FUNCTION "LHTTP_ExtractStringFromArray" : Word   // FC2, SCL
{ S7_Optimized_Access := 'TRUE' }
VERSION : 0.1
   VAR_INPUT
      textBefore : String;   // Text before text that is extracted
      textAfter : String;   // Text after text that is extracted
   END_VAR
   VAR_OUTPUT
      extractedString : String;   // Extracted string
   END_VAR
   VAR_IN_OUT
      searchIn : Array[*] of Char;   // Array of Char to search in
   END_VAR
   VAR_TEMP
      tempLowerBound : DInt;   // Lower bound of given array
      tempNumElements : UDInt;   // Number of elements in given array
      tempPosInArray : DInt;   // Position in array during search
      tempLenTextBefore : Int;   // Length of text before
      tempPosTextBefore : DInt;   // Position of text before in array of Char
      tempLenTextAfter : Int;   // Length of text after
      tempPosTextAfter : Int;   // Position of text after in converted string
      tempString : String;   // Temporary string to work with
   END_VAR
   // Ret_Val : Return value; 16#0000: Successful, text was found, 16#9001: Unsuccessful, only start text was found, extracted String is filled with characters after start text, 16#9002: Unsuccessful, neither text was found
   VAR CONSTANT
      LEN_STRING : UInt := 254;   // Max. length of String
      STATUS_TEXT_FOUND : Word := 16#0000;   // Texts before and after were found
      STATUS_ONLY_START : Word := 16#9001;   // Only text before was found
      STATUS_NOTHING_FOUND : Word := 16#9002;   // Neither text was found
   END_VAR
BEGIN
   //=============================================================================
   // SIEMENS AG
   // (c)Copyright 2019
   //-----------------------------------------------------------------------------
   // Library:       LHTTP
   // Tested with:   CPU 1516-3 PN/DP V2.6
   // Engineering:   TIA Portal V15.1
   // Restrictions:  --
   // Requirements:  --
   // Functionality: Extracts a String specified by a text before and after
   //                from an array of Char
   //-----------------------------------------------------------------------------
   // Change log table:
   // Version    Date         Expert in charge         Changes applied
   // 01.00.00   01.04.2019   Siemens Online Support   First released version
   //=============================================================================

   // Initialization
   #tempPosTextBefore := 0;
   #tempPosTextAfter := 0;
   #tempLenTextBefore := LEN(#textBefore);
   #tempLenTextAfter := LEN(#textAfter);
   #extractedString := '';
   #LHTTP_ExtractStringFromArray := #STATUS_NOTHING_FOUND;

   // Get number of elements
   #tempPosInArray := #tempLowerBound := LOWER_BOUND(ARR := #searchIn, DIM := 1);
   #tempNumElements := DINT_TO_UDINT(UPPER_BOUND(ARR := #searchIn, DIM := 1) - #tempLowerBound + 1);


   // Search for text before until something was found
   REPEAT

     // Convert Chars to String
     Chars_TO_Strg(Chars  := #searchIn,
                   pChars := #tempPosInArray - #tempLowerBound, // Subtract offset since pChars is zero based
                   Cnt    := UDINT_TO_UINT(MIN(IN1 := #LEN_STRING, IN2 := #tempNumElements)),
                   Strg   => #tempString);

     // Search for text before
     #tempPosTextBefore := FIND(IN1 := #tempString, IN2 := #textBefore);

     // Text before was found
     IF #tempPosTextBefore > 0 THEN

       // Set position in array to end of text before
       #tempPosInArray += #tempPosTextBefore + #tempLenTextBefore - 1;

       // Create new string from end of text before
       Chars_TO_Strg(Chars  := #searchIn,
                     pChars := #tempPosInArray - #tempLowerBound, // Subtract offset since pChars is zero based
                     Cnt    := UDINT_TO_UINT(MIN(IN1 := #LEN_STRING, IN2 := #tempNumElements)),
                     Strg   => #tempString);

       // Find end of string to be extracted
       #tempPosTextAfter := FIND(IN1 := #tempString, IN2 := #textAfter);

       IF #tempPosTextAfter > 0 THEN // Shorten string if text after was found

         #extractedString := LEFT(IN := #tempString, L := #tempPosTextAfter - 1);
         #LHTTP_ExtractStringFromArray := #STATUS_TEXT_FOUND;
         EXIT;

       ELSE // Output whole string if text after was not found

         #extractedString := #tempString;
         #LHTTP_ExtractStringFromArray := #STATUS_ONLY_START;
         EXIT;

       END_IF;

     ELSE
       // Otherwise continue search in next string minus length of text before to ensure
       // keywords are not broken up at the end of a string and thus missed
       #tempPosInArray += UINT_TO_INT(#LEN_STRING) - #tempLenTextBefore;
     END_IF;

     // Repeat until end of array is reached
   UNTIL (#tempPosInArray > #tempNumElements) END_REPEAT;
END_FUNCTION

FUNCTION "LHTTP_ExtractStringFromArrayExt" : Word   // FC4, SCL
{ S7_Optimized_Access := 'TRUE' }
VERSION : 0.1
   VAR_INPUT
      textBefore : String;   // Text before text that is extracted
      textAfter : String;   // Text after text that is extracted
      includeBeforeAfter : Bool;   // If TRUE, texts before and after are included in the extracted string
      startPos : DInt;   // Position within array to start search from
   END_VAR
   VAR_OUTPUT
      extractedString : String;   // Extracted string
      position : DInt;   // Position (index) within the array where text begins
      length : Int;   // Length of text that was extracted
   END_VAR
   VAR_IN_OUT
      searchIn : Array[*] of Char;   // Array of Char to search in
   END_VAR
   VAR_TEMP
      tempLowerBound : DInt;   // Lower bound of given array
      tempNumElements : UDInt;   // Number of elements in given array
      tempPosInArray : DInt;   // Position in array during search
      tempLenTextBefore : Int;   // Length of text before
      tempPosTextBefore : DInt;   // Position of text before in array of Char
      tempLenTextAfter : Int;   // Length of text after
      tempPosTextAfter : Int;   // Position of text after in converted string
      tempString : String;   // Temporary string to work with
   END_VAR
   // Ret_Val : Return value; 16#0000: Successful, text was found, 16#9001: Unsuccessful, only start text was found, extracted String is filled with characters after start text, 16#9002: Unsuccessful, neither text was found
   VAR CONSTANT
      LEN_STRING : UInt := 254;   // Max. length of String
      STATUS_TEXT_FOUND : Word := 16#0000;   // Start text and end text were found
      STATUS_ONLY_START : Word := 16#9001;   // Only start text was found
      STATUS_NOTHING_FOUND : Word := 16#9002;   // Neither text was found
   END_VAR
BEGIN
   //=============================================================================
   // SIEMENS AG
   // (c)Copyright 2019
   //-----------------------------------------------------------------------------
   // Library:       LHTTP
   // Tested with:   CPU 1516-3 PN/DP V2.6
   // Engineering:   TIA Portal V15.1
   // Restrictions:  --
   // Requirements:  --
   // Functionality: Extracts a String specified by a text before and after
   //                from an array of Char with extended options
   //-----------------------------------------------------------------------------
   // Change log table:
   // Version    Date         Expert in charge         Changes applied
   // 01.00.00   01.04.2019   Siemens Online Support   First released version
   //=============================================================================

   // Initialization
   #tempPosInArray := #startPos;
   #tempPosTextBefore := 0;
   #tempPosTextAfter := 0;
   #tempLenTextBefore := LEN(#textBefore);
   #tempLenTextAfter := LEN(#textAfter);
   #position := -1;
   #length := 0;
   #extractedString := '';
   #LHTTP_ExtractStringFromArrayExt := #STATUS_NOTHING_FOUND;

   // Get number of elements
   #tempLowerBound := LOWER_BOUND(ARR := #searchIn, DIM := 1);
   #tempNumElements := DINT_TO_UDINT(UPPER_BOUND(ARR := #searchIn, DIM := 1) - #tempLowerBound + 1);

   // Search for text before until something was found
   REPEAT

     // Convert Chars to String
     Chars_TO_Strg(Chars := #searchIn,
                   pChars := #tempPosInArray - #tempLowerBound, // Subtract offset since pChars is zero based
                   Cnt := UDINT_TO_UINT(MIN(IN1 := #LEN_STRING, IN2 := #tempNumElements)),
                   Strg => #tempString);

     // Search for text before
     #tempPosTextBefore := FIND(IN1 := #tempString, IN2 := #textBefore);

     // Text before was found
     IF #tempPosTextBefore > 0 THEN

       // Set position in array to beginning or end of text before
       IF #includeBeforeAfter THEN
         #tempPosInArray += #tempPosTextBefore - 1;
       ELSE
         #tempPosInArray += #tempPosTextBefore + #tempLenTextBefore - 1;
       END_IF;

       // Create new string from beginning or end of text before
       Chars_TO_Strg(Chars := #searchIn,
                     pChars := #tempPosInArray - #tempLowerBound, // Subtract offset since pChars is zero based
                     Cnt := UDINT_TO_UINT(MIN(IN1 := #LEN_STRING, IN2 := #tempNumElements)),
                     Strg => #tempString);

       // Find end of string to be extracted
       #tempPosTextAfter := FIND(IN1 := #tempString, IN2 := #textAfter);

       IF #tempPosTextAfter > 0 THEN // Shorten string if text after was found

         IF #includeBeforeAfter THEN
           #length := #tempPosTextAfter + #tempLenTextAfter - 1;
         ELSE
           #length := #tempPosTextAfter - 1;
         END_IF;

         #position := #tempPosInArray;
         #extractedString := LEFT(IN := #tempString, L := #length);
         #LHTTP_ExtractStringFromArrayExt := #STATUS_TEXT_FOUND;
         EXIT;

       ELSE // Output whole string if text after was not found

         #extractedString := #tempString;
         #position := #tempPosInArray;
         #length := LEN(#tempString);
         #LHTTP_ExtractStringFromArrayExt := #STATUS_ONLY_START;
         EXIT;

       END_IF;

     ELSE
       // Otherwise continue search in next string minus length of text before to ensure
       // keywords are not broken up at the end of a string and thus missed
       #tempPosInArray += UINT_TO_INT(#LEN_STRING) - #tempLenTextBefore;
     END_IF;

     // Repeat until end of array is reached
   UNTIL (#tempPosInArray > #tempNumElements) END_REPEAT;
END_FUNCTION

FUNCTION "LHTTP_FindStringInArray" : DInt   // FC5, SCL
{ S7_Optimized_Access := 'TRUE' }
VERSION : 0.1
   VAR_INPUT
      searchFor : String;   // Text that is searched for
   END_VAR
   VAR_IN_OUT
      searchIn : Array[*] of Char;   // Array of Char to search in
   END_VAR
   VAR_TEMP
      tempLowerBound : DInt;   // Lower bound of given array
      tempNumElements : UDInt;   // Number of elements in given array
      tempLenSearchFor : Int;   // Length of text that is seached for
      tempPosInArray : DInt;   // Position in array during search (0-based)
      tempPosInString : Int;   // Position in working string during search
      tempString : String;   // Temporary string to work with
   END_VAR
   // Ret_Val : Position (index) of the first character of the text that is searched for within the array of Char
   VAR CONSTANT
      LEN_STRING : UInt := 254;   // Max. length of String
   END_VAR
BEGIN
   //=============================================================================
   // SIEMENS AG
   // (c)Copyright 2019
   //-----------------------------------------------------------------------------
   // Library:       LHTTP
   // Tested with:   CPU 1516-3 PN/DP V2.6
   // Engineering:   TIA Portal V15.1
   // Restrictions:  --
   // Requirements:  --
   // Functionality: Searches for a specified String within an array of Char
   //-----------------------------------------------------------------------------
   // Change log table:
   // Version    Date         Expert in charge         Changes applied
   // 01.00.00   01.01.2019   Siemens Online Support   First released version
   //=============================================================================

   // Initialization
   #tempPosInString := 0;
   #tempPosInArray := 0;
   #tempLenSearchFor := LEN(#searchFor);
   #LHTTP_FindStringInArray := -1;

   // Get number of elements
   #tempLowerBound := LOWER_BOUND(ARR := #searchIn, DIM := 1);
   #tempNumElements := DINT_TO_UDINT(UPPER_BOUND(ARR := #searchIn, DIM := 1) - #tempLowerBound + 1);

   // Search for beginning of text until something was found
   REPEAT

     // Convert Chars to String
     Chars_TO_Strg(Chars := #searchIn,
                   pChars := #tempPosInArray,
                   Cnt := UDINT_TO_UINT(MIN(IN1 := #LEN_STRING, IN2 := #tempNumElements)),
                   Strg => #tempString);

     // Search for text at beginning
     #tempPosInString := FIND(IN1 := #tempString, IN2 := #searchFor);

     // Keyword was found
     IF #tempPosInString > 0 THEN
       // Output position of string
       #LHTTP_FindStringInArray := #tempLowerBound + #tempPosInArray + #tempPosInString - 1;
       EXIT;
     ELSE
       // Otherwise continue search in next string minus length of text at beginning to ensure
       // keywords are not broken up at the end of a string and thus missed
       #tempPosInArray += UINT_TO_INT(#LEN_STRING) - #tempLenSearchFor;
     END_IF;

   UNTIL (#tempPosInString > 0) OR (#tempPosInArray > #tempNumElements) END_REPEAT;
END_FUNCTION